PROGRAM MAIN
VAR CONSTANT
	iSoftMajorVersion			: INT	:= 2;
	iSoftMinorVersion			: INT	:= 0;

END_VAR
VAR PERSISTENT
	sMachineCnt					: TprodCounter;
	asStickData					: ARRAY[0..1] OF TStickData;
	asStickDataMMI				: ARRAY[0..1] OF TStickDataMMI;
	sStickDataShared			: TStickDataShared;
	sVacuumSettingsMMI			: TVacuumSettingsMMI;
	TAutoSampling				: TAutoSampling;
	bDisableCleanAfterPearling	: BOOL;
	bDisableVision				: BOOL;
	bSpeedModeSlow				: BOOL;
	iMachineWO					: DINT;
	iMachineSN					: INT;
END_VAR
VAR
	sMMI_SyncVar 				: TMachineData;			(* MMI interface data *)
	sMMI_ManualVar 				: TManualData;			(* MMI interface data for manual mode *)
	sMMI_VisionVar				: TVisionData;			(* Vision interface *)
	sMMI_ConfigFileData			: TConfigFileData;
	(* Blocks definitions *)
	TManager					: Manager;
	TLoaderHandler				: LoaderHdl;
	TTableHandler				: TableHdl;
	TPearlingHandler			: PearlingHdl;
	TSharpenHandler				: SharpenHdl;
	TTurnOverHandler			: TurnOverHdl;
	TBarrelHandler				: BarrelHdl;
	TLift1Handler				: LiftHdl;
	TLift2Handler				: LiftHdl;
	TRejectHandler				: RejectHdl;
	TVisionHandler				: VisionHdl;
	TUtilitiesHandler			: UtilitiesHdl;
	eBarrelCmd					: TModuleCommands;
	eLoaderCmd					: TModuleCommands;
	eTableCmd					: TModuleCommands;
	ePearlingCmd				: TModuleCommands;
	eSharpenCmd					: TModuleCommands;
	eTurnOverCmd				: TModuleCommands;
	eLift1Cmd					: TModuleCommands;
	eLift2Cmd					: TModuleCommands;
	eRejectCmd					: TModuleCommands;
	eVisionCmd					: TModuleCommands;
	eUtilitiesCmd				: TModuleCommands;
	TCheckDoors					: TON;
	sGiversTakers				: TStationGiversTakers;
	bFirstCycle					: BOOL				:= TRUE;
	bJobInProgress				: BOOL;
	bPearlingReady4ChangeTool	: BOOL;
	iStickArea2Use				: INT;
	bTableVacuuumNotOk			: BOOL;
	bPearlingHead1IsUsed		: BOOL;
	bPearlingHead2IsUsed		: BOOL;
	eTableSideForLoader			: TTableSide;
	sRunData					: TRunData;
	bTableAspiration13On		: BOOL;
	bTableAspiration24On		: BOOL;
	bLoaderBrushAspirationOn	: BOOL;
	bBrushAspirationOn			: BOOL;
	bSharpenAspirationOn		: BOOL;
	bStopRequest				: BOOL;
	bPauseRequest				: BOOL;
	bLayeringWithTwoParts		: BOOL;
	bNewPlateLift1				: BOOL;
	bNewPlateLift2				: BOOL;
	bNewPlateReject				: BOOL;
	bLoaderVacuumInUse			: BOOL;
	bManInterlockPearling		: BOOL;
	bManInterlockLoader			: BOOL;
	bManInterlockLoaderLift		: BOOL;
	bManInterlockTable			: BOOL;
	bManInterlockTurnOver		: BOOL;
	TJobElapsed					: TIME;
	aiTablePearlsVacuumFlow		: ARRAY[0..1] OF INT;
END_VAR
VAR // added by the converter: edge detectors and wires of the graphical bodies
    _w1, _w3 : TStickData;
    _w2, _w4 : TStickDataMMI;
    _w5 : TStickDataMMIShared;
    _w6 : TVacuumSettingsMMI;
    _w7 : TprodCounter;
    _w8, _w9, _w11, _w12 : INT;
    _w10, _w13, _w14, _w15 : BOOL;
END_VAR

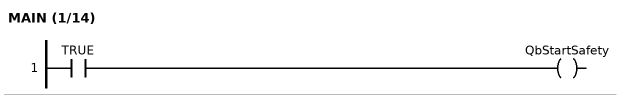
// NETWORK 1
QbStartSafety := TRUE;

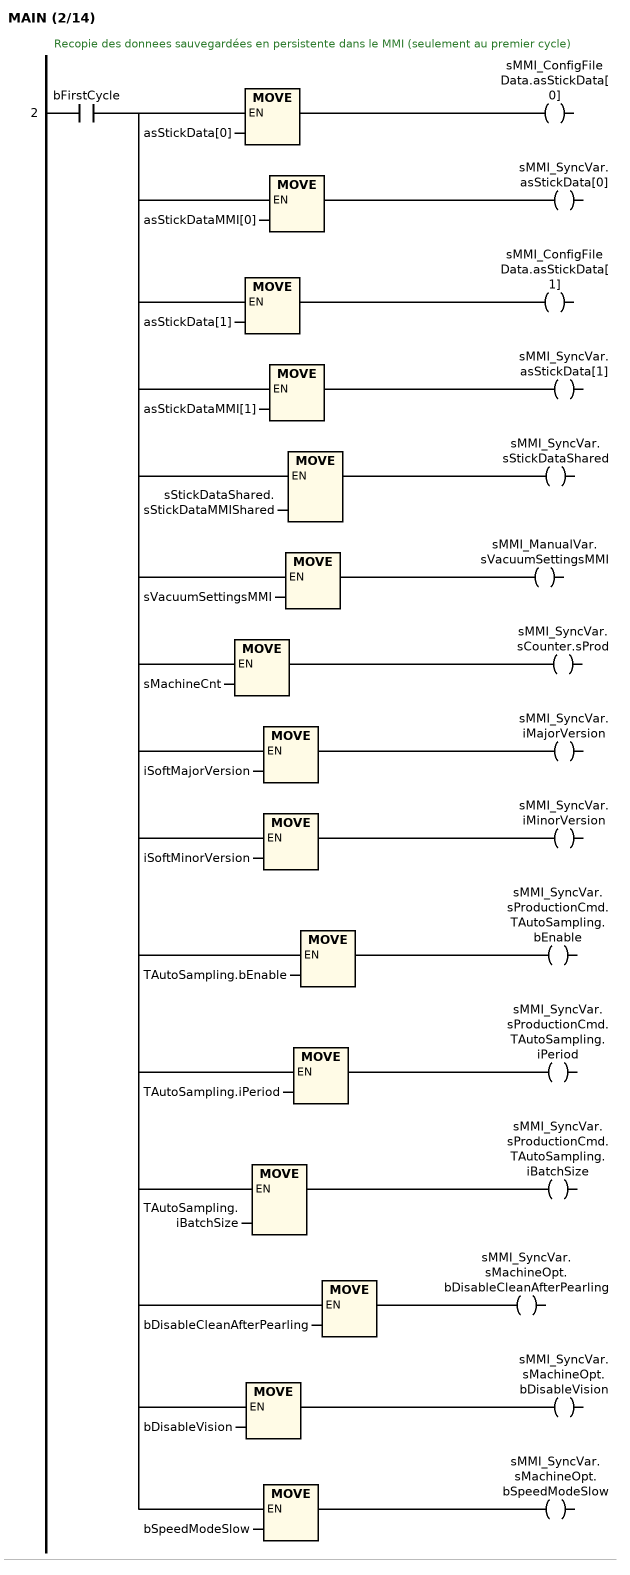
// NETWORK 2
// Recopie des donnees sauvegardées en persistente dans le MMI (seulement au premier cycle)
IF bFirstCycle THEN _w1 := asStickData[0]; END_IF
sMMI_ConfigFileData.asStickData[0] := _w1;
IF bFirstCycle THEN _w2 := asStickDataMMI[0]; END_IF
sMMI_SyncVar.asStickData[0] := _w2;
IF bFirstCycle THEN _w3 := asStickData[1]; END_IF
sMMI_ConfigFileData.asStickData[1] := _w3;
IF bFirstCycle THEN _w4 := asStickDataMMI[1]; END_IF
sMMI_SyncVar.asStickData[1] := _w4;
IF bFirstCycle THEN _w5 := sStickDataShared.sStickDataMMIShared; END_IF
sMMI_SyncVar.sStickDataShared := _w5;
IF bFirstCycle THEN _w6 := sVacuumSettingsMMI; END_IF
sMMI_ManualVar.sVacuumSettingsMMI := _w6;
IF bFirstCycle THEN _w7 := sMachineCnt; END_IF
sMMI_SyncVar.sCounter.sProd := _w7;
IF bFirstCycle THEN _w8 := iSoftMajorVersion; END_IF
sMMI_SyncVar.iMajorVersion := _w8;
IF bFirstCycle THEN _w9 := iSoftMinorVersion; END_IF
sMMI_SyncVar.iMinorVersion := _w9;
IF bFirstCycle THEN _w10 := TAutoSampling.bEnable; END_IF
sMMI_SyncVar.sProductionCmd.TAutoSampling.bEnable := _w10;
IF bFirstCycle THEN _w11 := TAutoSampling.iPeriod; END_IF
sMMI_SyncVar.sProductionCmd.TAutoSampling.iPeriod := _w11;
IF bFirstCycle THEN _w12 := TAutoSampling.iBatchSize; END_IF
sMMI_SyncVar.sProductionCmd.TAutoSampling.iBatchSize := _w12;
IF bFirstCycle THEN _w13 := bDisableCleanAfterPearling; END_IF
sMMI_SyncVar.sMachineOpt.bDisableCleanAfterPearling := _w13;
IF bFirstCycle THEN _w14 := bDisableVision; END_IF
sMMI_SyncVar.sMachineOpt.bDisableVision := _w14;
IF bFirstCycle THEN _w15 := bSpeedModeSlow; END_IF
sMMI_SyncVar.sMachineOpt.bSpeedModeSlow := _w15;

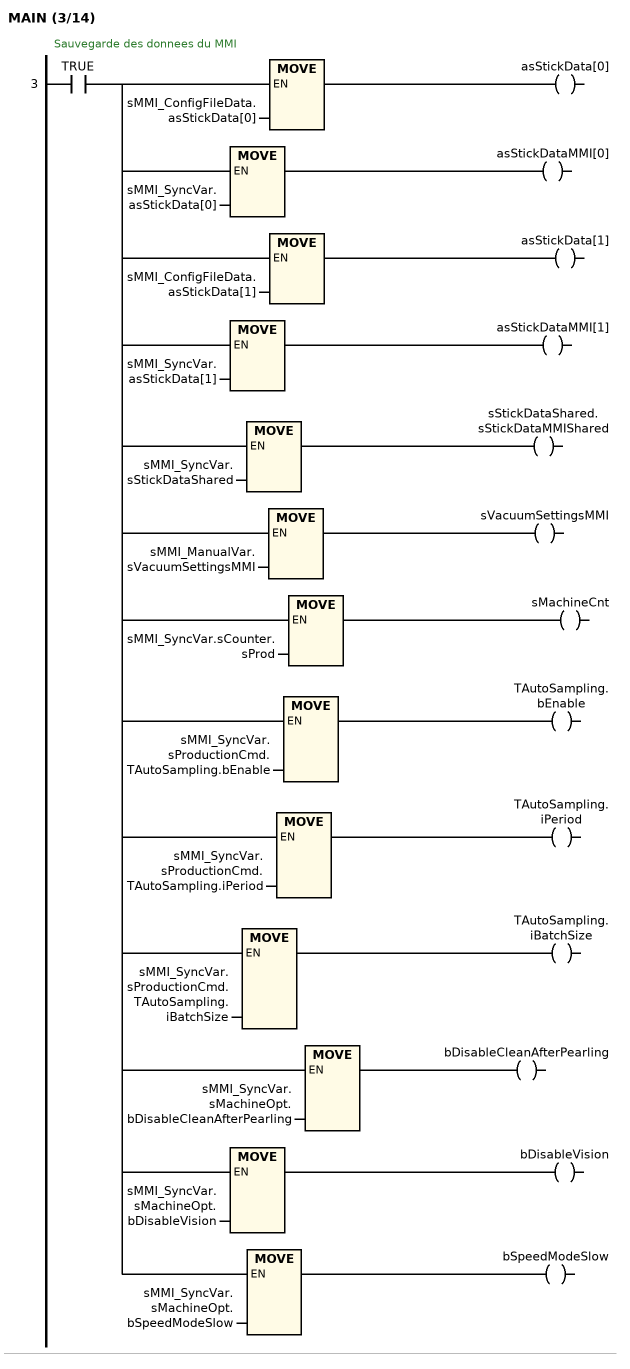
// NETWORK 3
// Sauvegarde des donnees du MMI
asStickData[0] := sMMI_ConfigFileData.asStickData[0];
asStickDataMMI[0] := sMMI_SyncVar.asStickData[0];
asStickData[1] := sMMI_ConfigFileData.asStickData[1];
asStickDataMMI[1] := sMMI_SyncVar.asStickData[1];
sStickDataShared.sStickDataMMIShared := sMMI_SyncVar.sStickDataShared;
sVacuumSettingsMMI := sMMI_ManualVar.sVacuumSettingsMMI;
sMachineCnt := sMMI_SyncVar.sCounter.sProd;
TAutoSampling.bEnable := sMMI_SyncVar.sProductionCmd.TAutoSampling.bEnable;
TAutoSampling.iPeriod := sMMI_SyncVar.sProductionCmd.TAutoSampling.iPeriod;
TAutoSampling.iBatchSize := sMMI_SyncVar.sProductionCmd.TAutoSampling.iBatchSize;
bDisableCleanAfterPearling := sMMI_SyncVar.sMachineOpt.bDisableCleanAfterPearling;
bDisableVision := sMMI_SyncVar.sMachineOpt.bDisableVision;
bSpeedModeSlow := sMMI_SyncVar.sMachineOpt.bSpeedModeSlow;

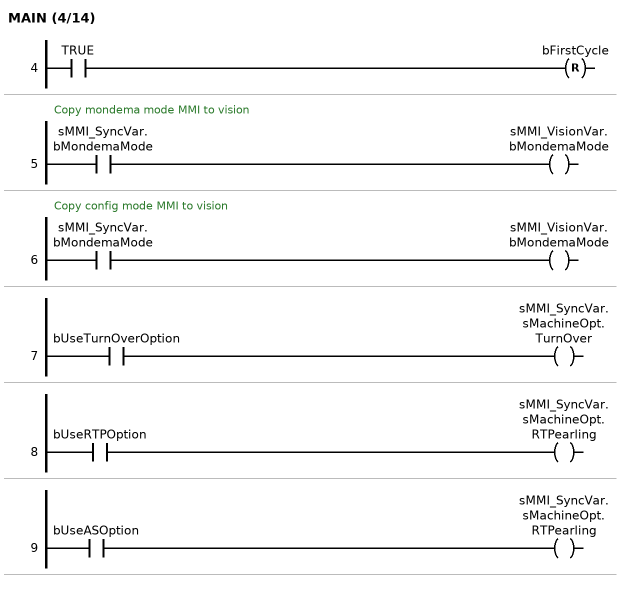
// NETWORK 4
bFirstCycle R= TRUE;

// NETWORK 5
// Copy mondema mode MMI to vision
sMMI_VisionVar.bMondemaMode := sMMI_SyncVar.bMondemaMode;

// NETWORK 6
// Copy config mode MMI to vision
sMMI_VisionVar.bMondemaMode := sMMI_SyncVar.bMondemaMode;

// NETWORK 7
sMMI_SyncVar.sMachineOpt.TurnOver := bUseTurnOverOption;

// NETWORK 8
sMMI_SyncVar.sMachineOpt.RTPearling := bUseRTPOption;

// NETWORK 9
sMMI_SyncVar.sMachineOpt.RTPearling := bUseASOption;

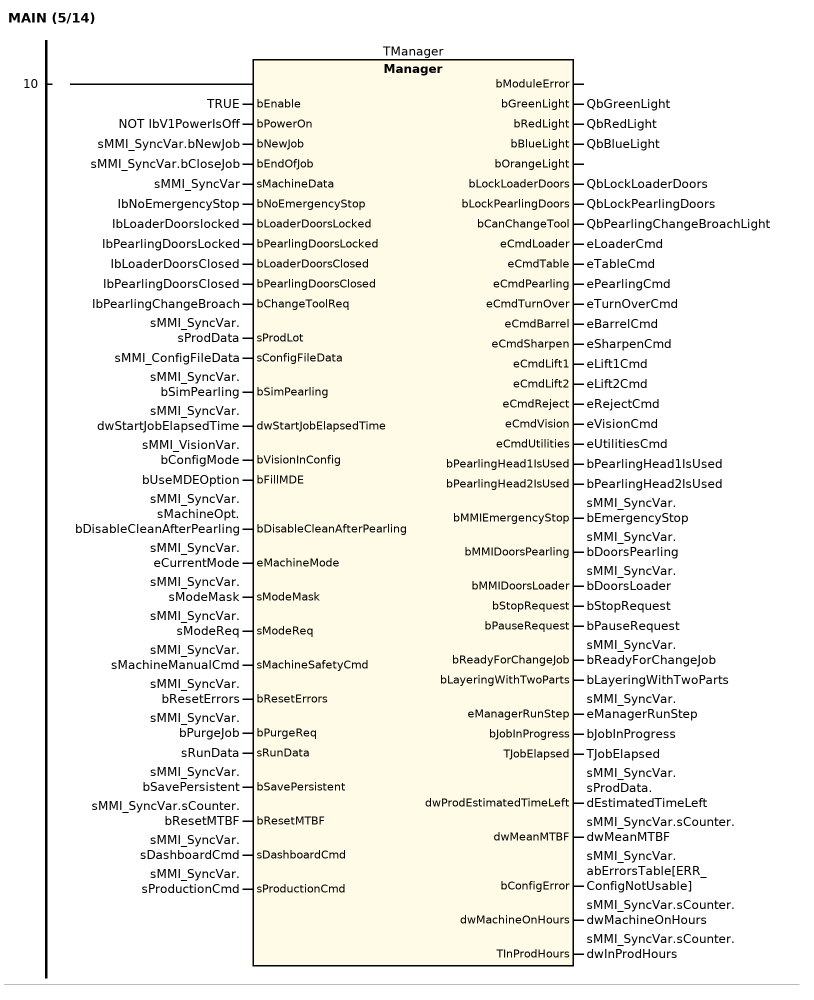
// NETWORK 10
TManager(
    bEnable := TRUE,
    bPowerOn := NOT IbV1PowerIsOff,
    bNewJob := sMMI_SyncVar.bNewJob,
    bEndOfJob := sMMI_SyncVar.bCloseJob,
    sMachineData := sMMI_SyncVar,
    bNoEmergencyStop := IbNoEmergencyStop,
    bLoaderDoorsLocked := IbLoaderDoorslocked,
    bPearlingDoorsLocked := IbPearlingDoorsLocked,
    bLoaderDoorsClosed := IbLoaderDoorsClosed,
    bPearlingDoorsClosed := IbPearlingDoorsClosed,
    bChangeToolReq := IbPearlingChangeBroach,
    sProdLot := sMMI_SyncVar.sProdData,
    sConfigFileData := sMMI_ConfigFileData,
    bSimPearling := sMMI_SyncVar.bSimPearling,
    dwStartJobElapsedTime := sMMI_SyncVar.dwStartJobElapsedTime,
    bVisionInConfig := sMMI_VisionVar.bConfigMode,
    bFillMDE := bUseMDEOption,
    bDisableCleanAfterPearling := sMMI_SyncVar.sMachineOpt.bDisableCleanAfterPearling,
    eMachineMode := sMMI_SyncVar.eCurrentMode,
    sModeMask := sMMI_SyncVar.sModeMask,
    sModeReq := sMMI_SyncVar.sModeReq,
    sMachineSafetyCmd := sMMI_SyncVar.sMachineManualCmd,
    bResetErrors := sMMI_SyncVar.bResetErrors,
    bPurgeReq := sMMI_SyncVar.bPurgeJob,
    sRunData := sRunData,
    bSavePersistent := sMMI_SyncVar.bSavePersistent,
    bResetMTBF := sMMI_SyncVar.sCounter.bResetMTBF,
    sDashboardCmd := sMMI_SyncVar.sDashboardCmd,
    sProductionCmd := sMMI_SyncVar.sProductionCmd,
    bGreenLight => QbGreenLight,
    bRedLight => QbRedLight,
    bBlueLight => QbBlueLight,
    bLockLoaderDoors => QbLockLoaderDoors,
    bLockPearlingDoors => QbLockPearlingDoors,
    bCanChangeTool => QbPearlingChangeBroachLight,
    eCmdLoader => eLoaderCmd,
    eCmdTable => eTableCmd,
    eCmdPearling => ePearlingCmd,
    eCmdTurnOver => eTurnOverCmd,
    eCmdBarrel => eBarrelCmd,
    eCmdSharpen => eSharpenCmd,
    eCmdLift1 => eLift1Cmd,
    eCmdLift2 => eLift2Cmd,
    eCmdReject => eRejectCmd,
    eCmdVision => eVisionCmd,
    eCmdUtilities => eUtilitiesCmd,
    bPearlingHead1IsUsed => bPearlingHead1IsUsed,
    bPearlingHead2IsUsed => bPearlingHead2IsUsed,
    bMMIEmergencyStop => sMMI_SyncVar.bEmergencyStop,
    bMMIDoorsPearling => sMMI_SyncVar.bDoorsPearling,
    bMMIDoorsLoader => sMMI_SyncVar.bDoorsLoader,
    bStopRequest => bStopRequest,
    bPauseRequest => bPauseRequest,
    bReadyForChangeJob => sMMI_SyncVar.bReadyForChangeJob,
    bLayeringWithTwoParts => bLayeringWithTwoParts,
    eManagerRunStep => sMMI_SyncVar.eManagerRunStep,
    bJobInProgress => bJobInProgress,
    TJobElapsed => TJobElapsed,
    dwProdEstimatedTimeLeft => sMMI_SyncVar.sProdData.dEstimatedTimeLeft,
    dwMeanMTBF => sMMI_SyncVar.sCounter.dwMeanMTBF,
    bConfigError => sMMI_SyncVar.abErrorsTable[ERR_ConfigNotUsable],
    dwMachineOnHours => sMMI_SyncVar.sCounter.dwMachineOnHours,
    TInProdHours => sMMI_SyncVar.sCounter.dwInProdHours); // Manager

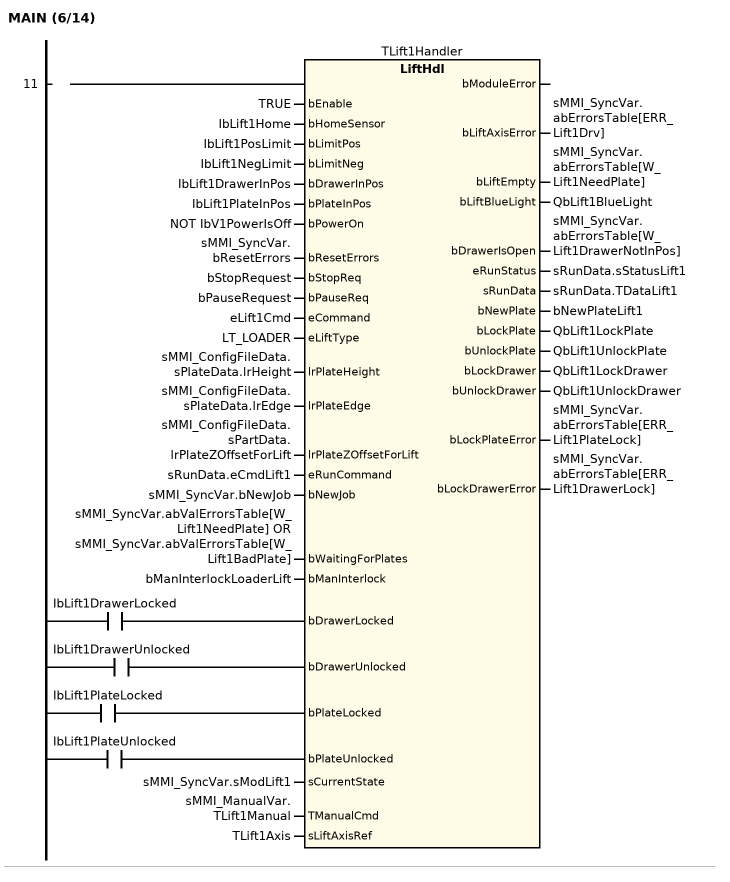
// NETWORK 11
TLift1Handler(
    bEnable := TRUE,
    bHomeSensor := IbLift1Home,
    bLimitPos := IbLift1PosLimit,
    bLimitNeg := IbLift1NegLimit,
    bDrawerInPos := IbLift1DrawerInPos,
    bPlateInPos := IbLift1PlateInPos,
    bPowerOn := NOT IbV1PowerIsOff,
    bResetErrors := sMMI_SyncVar.bResetErrors,
    bStopReq := bStopRequest,
    bPauseReq := bPauseRequest,
    eCommand := eLift1Cmd,
    eLiftType := LT_LOADER,
    lrPlateHeight := sMMI_ConfigFileData.sPlateData.lrHeight,
    lrPlateEdge := sMMI_ConfigFileData.sPlateData.lrEdge,
    lrPlateZOffsetForLift := sMMI_ConfigFileData.sPartData.lrPlateZOffsetForLift,
    eRunCommand := sRunData.eCmdLift1,
    bNewJob := sMMI_SyncVar.bNewJob,
    bWaitingForPlates := sMMI_SyncVar.abValErrorsTable[W_Lift1NeedPlate] OR sMMI_SyncVar.abValErrorsTable[W_Lift1BadPlate],
    bManInterlock := bManInterlockLoaderLift,
    bDrawerLocked := IbLift1DrawerLocked,
    bDrawerUnlocked := IbLift1DrawerUnlocked,
    bPlateLocked := IbLift1PlateLocked,
    bPlateUnlocked := IbLift1PlateUnlocked,
    sCurrentState := sMMI_SyncVar.sModLift1,
    TManualCmd := sMMI_ManualVar.TLift1Manual,
    sLiftAxisRef := TLift1Axis,
    bLiftAxisError => sMMI_SyncVar.abErrorsTable[ERR_Lift1Drv],
    bLiftEmpty => sMMI_SyncVar.abErrorsTable[W_Lift1NeedPlate],
    bLiftBlueLight => QbLift1BlueLight,
    bDrawerIsOpen => sMMI_SyncVar.abErrorsTable[W_Lift1DrawerNotInPos],
    eRunStatus => sRunData.sStatusLift1,
    sRunData => sRunData.TDataLift1,
    bNewPlate => bNewPlateLift1,
    bLockPlate => QbLift1LockPlate,
    bUnlockPlate => QbLift1UnlockPlate,
    bLockDrawer => QbLift1LockDrawer,
    bUnlockDrawer => QbLift1UnlockDrawer,
    bLockPlateError => sMMI_SyncVar.abErrorsTable[ERR_Lift1PlateLock],
    bLockDrawerError => sMMI_SyncVar.abErrorsTable[ERR_Lift1DrawerLock]); // LiftHdl

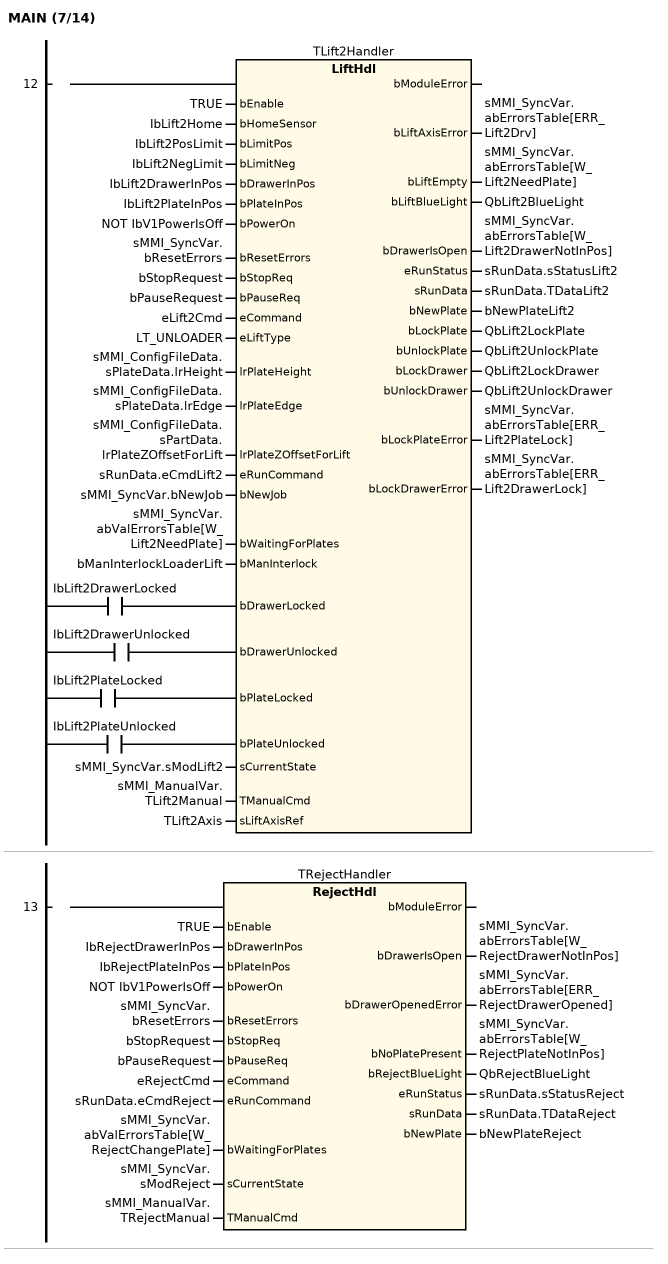
// NETWORK 12
TLift2Handler(
    bEnable := TRUE,
    bHomeSensor := IbLift2Home,
    bLimitPos := IbLift2PosLimit,
    bLimitNeg := IbLift2NegLimit,
    bDrawerInPos := IbLift2DrawerInPos,
    bPlateInPos := IbLift2PlateInPos,
    bPowerOn := NOT IbV1PowerIsOff,
    bResetErrors := sMMI_SyncVar.bResetErrors,
    bStopReq := bStopRequest,
    bPauseReq := bPauseRequest,
    eCommand := eLift2Cmd,
    eLiftType := LT_UNLOADER,
    lrPlateHeight := sMMI_ConfigFileData.sPlateData.lrHeight,
    lrPlateEdge := sMMI_ConfigFileData.sPlateData.lrEdge,
    lrPlateZOffsetForLift := sMMI_ConfigFileData.sPartData.lrPlateZOffsetForLift,
    eRunCommand := sRunData.eCmdLift2,
    bNewJob := sMMI_SyncVar.bNewJob,
    bWaitingForPlates := sMMI_SyncVar.abValErrorsTable[W_Lift2NeedPlate],
    bManInterlock := bManInterlockLoaderLift,
    bDrawerLocked := IbLift2DrawerLocked,
    bDrawerUnlocked := IbLift2DrawerUnlocked,
    bPlateLocked := IbLift2PlateLocked,
    bPlateUnlocked := IbLift2PlateUnlocked,
    sCurrentState := sMMI_SyncVar.sModLift2,
    TManualCmd := sMMI_ManualVar.TLift2Manual,
    sLiftAxisRef := TLift2Axis,
    bLiftAxisError => sMMI_SyncVar.abErrorsTable[ERR_Lift2Drv],
    bLiftEmpty => sMMI_SyncVar.abErrorsTable[W_Lift2NeedPlate],
    bLiftBlueLight => QbLift2BlueLight,
    bDrawerIsOpen => sMMI_SyncVar.abErrorsTable[W_Lift2DrawerNotInPos],
    eRunStatus => sRunData.sStatusLift2,
    sRunData => sRunData.TDataLift2,
    bNewPlate => bNewPlateLift2,
    bLockPlate => QbLift2LockPlate,
    bUnlockPlate => QbLift2UnlockPlate,
    bLockDrawer => QbLift2LockDrawer,
    bUnlockDrawer => QbLift2UnlockDrawer,
    bLockPlateError => sMMI_SyncVar.abErrorsTable[ERR_Lift2PlateLock],
    bLockDrawerError => sMMI_SyncVar.abErrorsTable[ERR_Lift2DrawerLock]); // LiftHdl

// NETWORK 13
TRejectHandler(
    bEnable := TRUE,
    bDrawerInPos := IbRejectDrawerInPos,
    bPlateInPos := IbRejectPlateInPos,
    bPowerOn := NOT IbV1PowerIsOff,
    bResetErrors := sMMI_SyncVar.bResetErrors,
    bStopReq := bStopRequest,
    bPauseReq := bPauseRequest,
    eCommand := eRejectCmd,
    eRunCommand := sRunData.eCmdReject,
    bWaitingForPlates := sMMI_SyncVar.abValErrorsTable[W_RejectChangePlate],
    sCurrentState := sMMI_SyncVar.sModReject,
    TManualCmd := sMMI_ManualVar.TRejectManual,
    bDrawerIsOpen => sMMI_SyncVar.abErrorsTable[W_RejectDrawerNotInPos],
    bDrawerOpenedError => sMMI_SyncVar.abErrorsTable[ERR_RejectDrawerOpened],
    bNoPlatePresent => sMMI_SyncVar.abErrorsTable[W_RejectPlateNotInPos],
    bRejectBlueLight => QbRejectBlueLight,
    eRunStatus => sRunData.sStatusReject,
    sRunData => sRunData.TDataReject,
    bNewPlate => bNewPlateReject); // RejectHdl

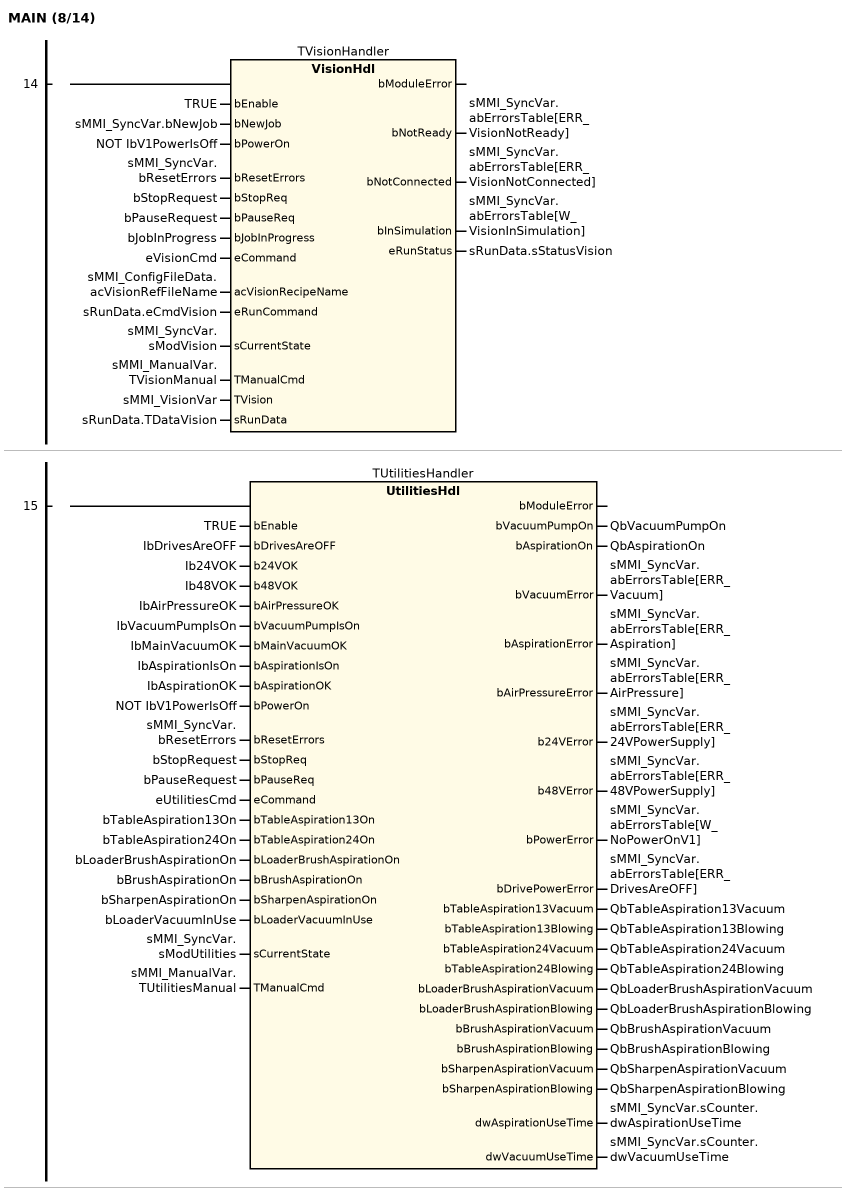
// NETWORK 14
TVisionHandler(
    bEnable := TRUE,
    bNewJob := sMMI_SyncVar.bNewJob,
    bPowerOn := NOT IbV1PowerIsOff,
    bResetErrors := sMMI_SyncVar.bResetErrors,
    bStopReq := bStopRequest,
    bPauseReq := bPauseRequest,
    bJobInProgress := bJobInProgress,
    eCommand := eVisionCmd,
    acVisionRecipeName := sMMI_ConfigFileData.acVisionRefFileName,
    eRunCommand := sRunData.eCmdVision,
    sCurrentState := sMMI_SyncVar.sModVision,
    TManualCmd := sMMI_ManualVar.TVisionManual,
    TVision := sMMI_VisionVar,
    sRunData := sRunData.TDataVision,
    bNotReady => sMMI_SyncVar.abErrorsTable[ERR_VisionNotReady],
    bNotConnected => sMMI_SyncVar.abErrorsTable[ERR_VisionNotConnected],
    bInSimulation => sMMI_SyncVar.abErrorsTable[W_VisionInSimulation],
    eRunStatus => sRunData.sStatusVision); // VisionHdl

// NETWORK 15
TUtilitiesHandler(
    bEnable := TRUE,
    bDrivesAreOFF := IbDrivesAreOFF,
    b24VOK := Ib24VOK,
    b48VOK := Ib48VOK,
    bAirPressureOK := IbAirPressureOK,
    bVacuumPumpIsOn := IbVacuumPumpIsOn,
    bMainVacuumOK := IbMainVacuumOK,
    bAspirationIsOn := IbAspirationIsOn,
    bAspirationOK := IbAspirationOK,
    bPowerOn := NOT IbV1PowerIsOff,
    bResetErrors := sMMI_SyncVar.bResetErrors,
    bStopReq := bStopRequest,
    bPauseReq := bPauseRequest,
    eCommand := eUtilitiesCmd,
    bTableAspiration13On := bTableAspiration13On,
    bTableAspiration24On := bTableAspiration24On,
    bLoaderBrushAspirationOn := bLoaderBrushAspirationOn,
    bBrushAspirationOn := bBrushAspirationOn,
    bSharpenAspirationOn := bSharpenAspirationOn,
    bLoaderVacuumInUse := bLoaderVacuumInUse,
    sCurrentState := sMMI_SyncVar.sModUtilities,
    TManualCmd := sMMI_ManualVar.TUtilitiesManual,
    bVacuumPumpOn => QbVacuumPumpOn,
    bAspirationOn => QbAspirationOn,
    bVacuumError => sMMI_SyncVar.abErrorsTable[ERR_Vacuum],
    bAspirationError => sMMI_SyncVar.abErrorsTable[ERR_Aspiration],
    bAirPressureError => sMMI_SyncVar.abErrorsTable[ERR_AirPressure],
    b24VError => sMMI_SyncVar.abErrorsTable[ERR_24VPowerSupply],
    b48VError => sMMI_SyncVar.abErrorsTable[ERR_48VPowerSupply],
    bPowerError => sMMI_SyncVar.abErrorsTable[W_NoPowerOnV1],
    bDrivePowerError => sMMI_SyncVar.abErrorsTable[ERR_DrivesAreOFF],
    bTableAspiration13Vacuum => QbTableAspiration13Vacuum,
    bTableAspiration13Blowing => QbTableAspiration13Blowing,
    bTableAspiration24Vacuum => QbTableAspiration24Vacuum,
    bTableAspiration24Blowing => QbTableAspiration24Blowing,
    bLoaderBrushAspirationVacuum => QbLoaderBrushAspirationVacuum,
    bLoaderBrushAspirationBlowing => QbLoaderBrushAspirationBlowing,
    bBrushAspirationVacuum => QbBrushAspirationVacuum,
    bBrushAspirationBlowing => QbBrushAspirationBlowing,
    bSharpenAspirationVacuum => QbSharpenAspirationVacuum,
    bSharpenAspirationBlowing => QbSharpenAspirationBlowing,
    dwAspirationUseTime => sMMI_SyncVar.sCounter.dwAspirationUseTime,
    dwVacuumUseTime => sMMI_SyncVar.sCounter.dwVacuumUseTime); // UtilitiesHdl

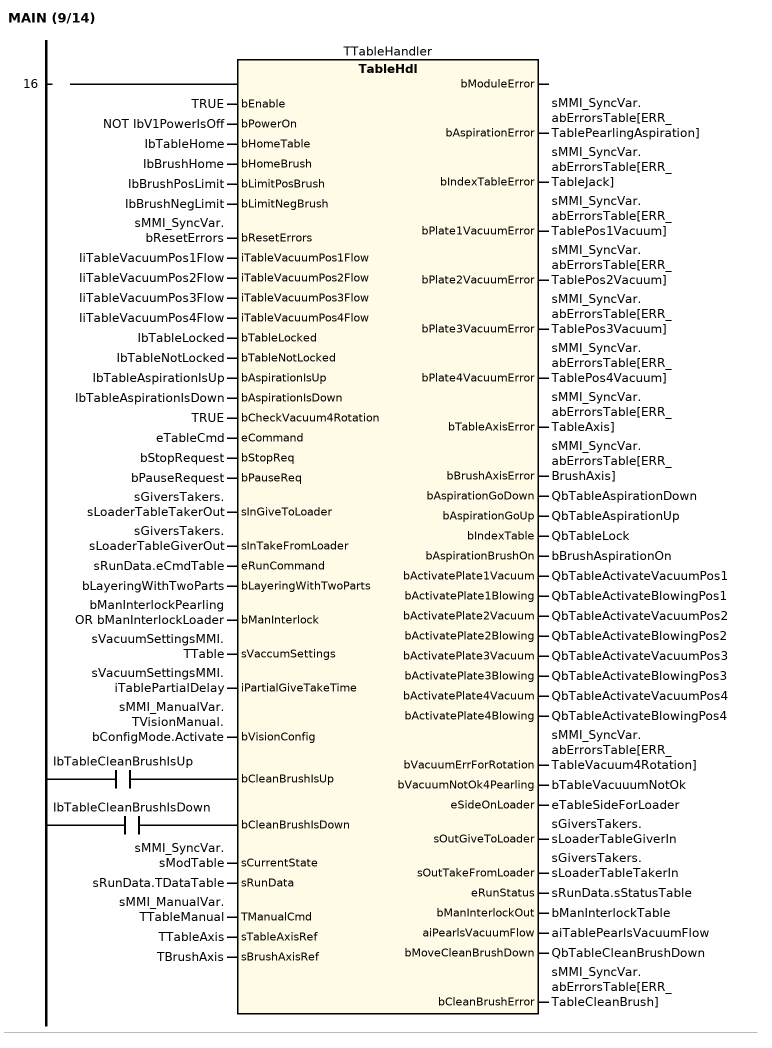
// NETWORK 16
TTableHandler(
    bEnable := TRUE,
    bPowerOn := NOT IbV1PowerIsOff,
    bHomeTable := IbTableHome,
    bHomeBrush := IbBrushHome,
    bLimitPosBrush := IbBrushPosLimit,
    bLimitNegBrush := IbBrushNegLimit,
    bResetErrors := sMMI_SyncVar.bResetErrors,
    iTableVacuumPos1Flow := IiTableVacuumPos1Flow,
    iTableVacuumPos2Flow := IiTableVacuumPos2Flow,
    iTableVacuumPos3Flow := IiTableVacuumPos3Flow,
    iTableVacuumPos4Flow := IiTableVacuumPos4Flow,
    bTableLocked := IbTableLocked,
    bTableNotLocked := IbTableNotLocked,
    bAspirationIsUp := IbTableAspirationIsUp,
    bAspirationIsDown := IbTableAspirationIsDown,
    bCheckVacuum4Rotation := TRUE,
    eCommand := eTableCmd,
    bStopReq := bStopRequest,
    bPauseReq := bPauseRequest,
    sInGiveToLoader := sGiversTakers.sLoaderTableTakerOut,
    sInTakeFromLoader := sGiversTakers.sLoaderTableGiverOut,
    eRunCommand := sRunData.eCmdTable,
    bLayeringWithTwoParts := bLayeringWithTwoParts,
    bManInterlock := bManInterlockPearling OR bManInterlockLoader,
    sVaccumSettings := sVacuumSettingsMMI.TTable,
    iPartialGiveTakeTime := sVacuumSettingsMMI.iTablePartialDelay,
    bVisionConfig := sMMI_ManualVar.TVisionManual.bConfigMode.Activate,
    bCleanBrushIsUp := IbTableCleanBrushIsUp,
    bCleanBrushIsDown := IbTableCleanBrushIsDown,
    sCurrentState := sMMI_SyncVar.sModTable,
    sRunData := sRunData.TDataTable,
    TManualCmd := sMMI_ManualVar.TTableManual,
    sTableAxisRef := TTableAxis,
    sBrushAxisRef := TBrushAxis,
    bAspirationError => sMMI_SyncVar.abErrorsTable[ERR_TablePearlingAspiration],
    bIndexTableError => sMMI_SyncVar.abErrorsTable[ERR_TableJack],
    bPlate1VacuumError => sMMI_SyncVar.abErrorsTable[ERR_TablePos1Vacuum],
    bPlate2VacuumError => sMMI_SyncVar.abErrorsTable[ERR_TablePos2Vacuum],
    bPlate3VacuumError => sMMI_SyncVar.abErrorsTable[ERR_TablePos3Vacuum],
    bPlate4VacuumError => sMMI_SyncVar.abErrorsTable[ERR_TablePos4Vacuum],
    bTableAxisError => sMMI_SyncVar.abErrorsTable[ERR_TableAxis],
    bBrushAxisError => sMMI_SyncVar.abErrorsTable[ERR_BrushAxis],
    bAspirationGoDown => QbTableAspirationDown,
    bAspirationGoUp => QbTableAspirationUp,
    bIndexTable => QbTableLock,
    bAspirationBrushOn => bBrushAspirationOn,
    bActivatePlate1Vacuum => QbTableActivateVacuumPos1,
    bActivatePlate1Blowing => QbTableActivateBlowingPos1,
    bActivatePlate2Vacuum => QbTableActivateVacuumPos2,
    bActivatePlate2Blowing => QbTableActivateBlowingPos2,
    bActivatePlate3Vacuum => QbTableActivateVacuumPos3,
    bActivatePlate3Blowing => QbTableActivateBlowingPos3,
    bActivatePlate4Vacuum => QbTableActivateVacuumPos4,
    bActivatePlate4Blowing => QbTableActivateBlowingPos4,
    bVacuumErrForRotation => sMMI_SyncVar.abErrorsTable[ERR_TableVacuum4Rotation],
    bVacuumNotOk4Pearling => bTableVacuuumNotOk,
    eSideOnLoader => eTableSideForLoader,
    sOutGiveToLoader => sGiversTakers.sLoaderTableGiverIn,
    sOutTakeFromLoader => sGiversTakers.sLoaderTableTakerIn,
    eRunStatus => sRunData.sStatusTable,
    bManInterlockOut => bManInterlockTable,
    aiPearlsVacuumFlow => aiTablePearlsVacuumFlow,
    bMoveCleanBrushDown => QbTableCleanBrushDown,
    bCleanBrushError => sMMI_SyncVar.abErrorsTable[ERR_TableCleanBrush]); // TableHdl

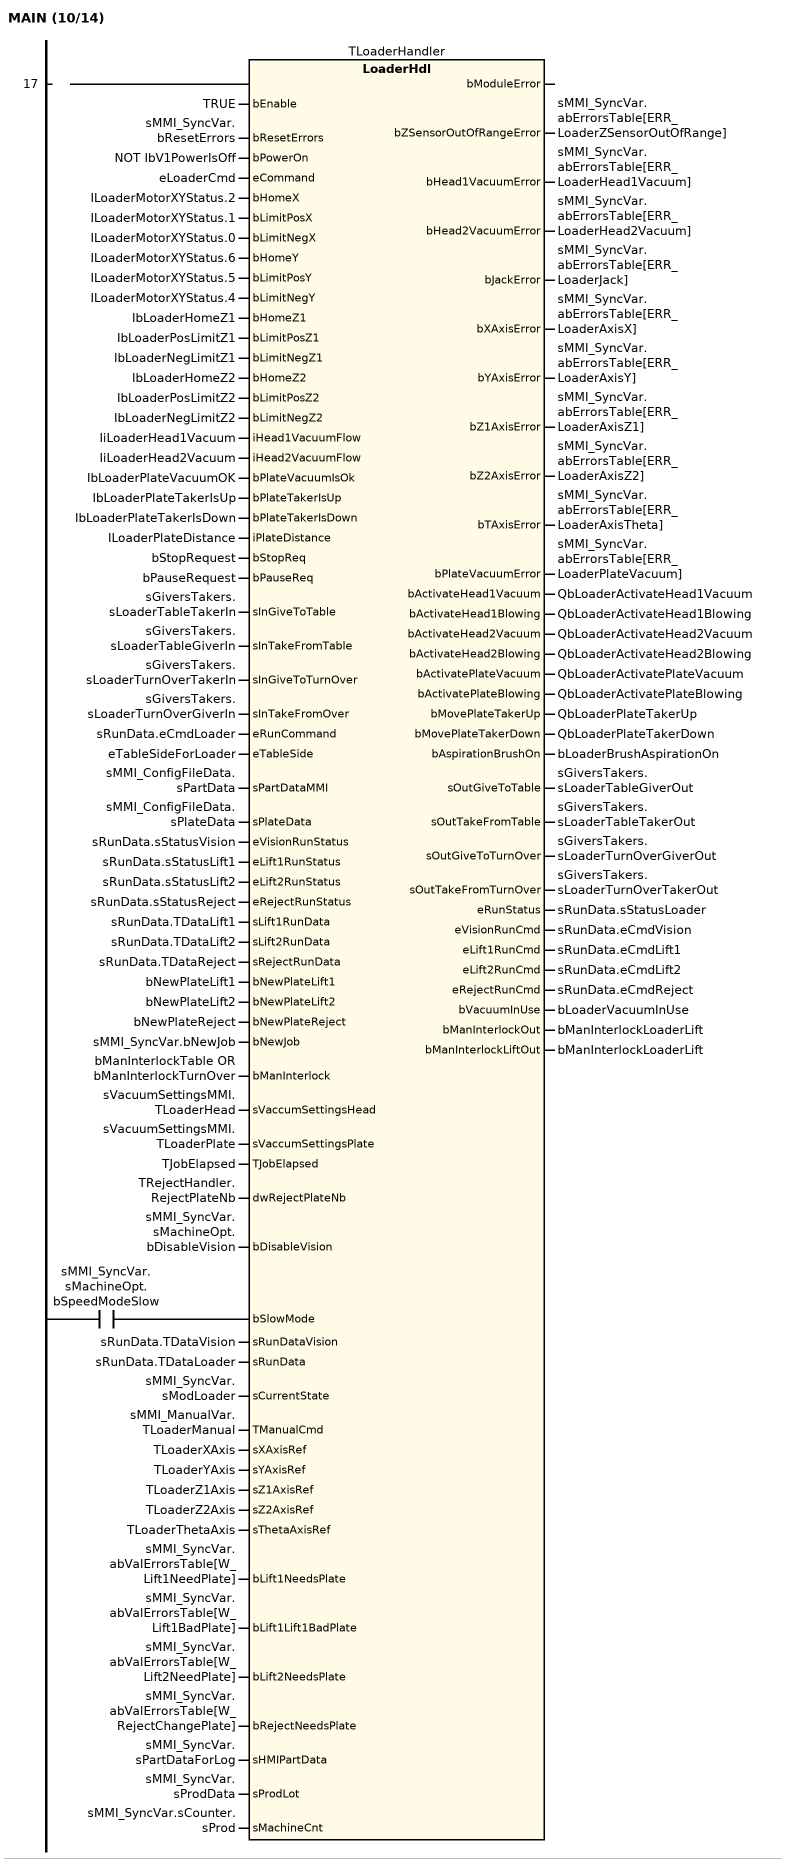
// NETWORK 17
TLoaderHandler(
    bEnable := TRUE,
    bResetErrors := sMMI_SyncVar.bResetErrors,
    bPowerOn := NOT IbV1PowerIsOff,
    eCommand := eLoaderCmd,
    bHomeX := ILoaderMotorXYStatus.2,
    bLimitPosX := ILoaderMotorXYStatus.1,
    bLimitNegX := ILoaderMotorXYStatus.0,
    bHomeY := ILoaderMotorXYStatus.6,
    bLimitPosY := ILoaderMotorXYStatus.5,
    bLimitNegY := ILoaderMotorXYStatus.4,
    bHomeZ1 := IbLoaderHomeZ1,
    bLimitPosZ1 := IbLoaderPosLimitZ1,
    bLimitNegZ1 := IbLoaderNegLimitZ1,
    bHomeZ2 := IbLoaderHomeZ2,
    bLimitPosZ2 := IbLoaderPosLimitZ2,
    bLimitNegZ2 := IbLoaderNegLimitZ2,
    iHead1VacuumFlow := IiLoaderHead1Vacuum,
    iHead2VacuumFlow := IiLoaderHead2Vacuum,
    bPlateVacuumIsOk := IbLoaderPlateVacuumOK,
    bPlateTakerIsUp := IbLoaderPlateTakerIsUp,
    bPlateTakerIsDown := IbLoaderPlateTakerIsDown,
    iPlateDistance := ILoaderPlateDistance,
    bStopReq := bStopRequest,
    bPauseReq := bPauseRequest,
    sInGiveToTable := sGiversTakers.sLoaderTableTakerIn,
    sInTakeFromTable := sGiversTakers.sLoaderTableGiverIn,
    sInGiveToTurnOver := sGiversTakers.sLoaderTurnOverTakerIn,
    sInTakeFromOver := sGiversTakers.sLoaderTurnOverGiverIn,
    eRunCommand := sRunData.eCmdLoader,
    eTableSide := eTableSideForLoader,
    sPartDataMMI := sMMI_ConfigFileData.sPartData,
    sPlateData := sMMI_ConfigFileData.sPlateData,
    eVisionRunStatus := sRunData.sStatusVision,
    eLift1RunStatus := sRunData.sStatusLift1,
    eLift2RunStatus := sRunData.sStatusLift2,
    eRejectRunStatus := sRunData.sStatusReject,
    sLift1RunData := sRunData.TDataLift1,
    sLift2RunData := sRunData.TDataLift2,
    sRejectRunData := sRunData.TDataReject,
    bNewPlateLift1 := bNewPlateLift1,
    bNewPlateLift2 := bNewPlateLift2,
    bNewPlateReject := bNewPlateReject,
    bNewJob := sMMI_SyncVar.bNewJob,
    bManInterlock := bManInterlockTable OR bManInterlockTurnOver,
    sVaccumSettingsHead := sVacuumSettingsMMI.TLoaderHead,
    sVaccumSettingsPlate := sVacuumSettingsMMI.TLoaderPlate,
    TJobElapsed := TJobElapsed,
    dwRejectPlateNb := TRejectHandler.RejectPlateNb,
    bDisableVision := sMMI_SyncVar.sMachineOpt.bDisableVision,
    bSlowMode := sMMI_SyncVar.sMachineOpt.bSpeedModeSlow,
    sRunDataVision := sRunData.TDataVision,
    sRunData := sRunData.TDataLoader,
    sCurrentState := sMMI_SyncVar.sModLoader,
    TManualCmd := sMMI_ManualVar.TLoaderManual,
    sXAxisRef := TLoaderXAxis,
    sYAxisRef := TLoaderYAxis,
    sZ1AxisRef := TLoaderZ1Axis,
    sZ2AxisRef := TLoaderZ2Axis,
    sThetaAxisRef := TLoaderThetaAxis,
    bLift1NeedsPlate := sMMI_SyncVar.abValErrorsTable[W_Lift1NeedPlate],
    bLift1Lift1BadPlate := sMMI_SyncVar.abValErrorsTable[W_Lift1BadPlate],
    bLift2NeedsPlate := sMMI_SyncVar.abValErrorsTable[W_Lift2NeedPlate],
    bRejectNeedsPlate := sMMI_SyncVar.abValErrorsTable[W_RejectChangePlate],
    sHMIPartData := sMMI_SyncVar.sPartDataForLog,
    sProdLot := sMMI_SyncVar.sProdData,
    sMachineCnt := sMMI_SyncVar.sCounter.sProd,
    bZSensorOutOfRangeError => sMMI_SyncVar.abErrorsTable[ERR_LoaderZSensorOutOfRange],
    bHead1VacuumError => sMMI_SyncVar.abErrorsTable[ERR_LoaderHead1Vacuum],
    bHead2VacuumError => sMMI_SyncVar.abErrorsTable[ERR_LoaderHead2Vacuum],
    bJackError => sMMI_SyncVar.abErrorsTable[ERR_LoaderJack],
    bXAxisError => sMMI_SyncVar.abErrorsTable[ERR_LoaderAxisX],
    bYAxisError => sMMI_SyncVar.abErrorsTable[ERR_LoaderAxisY],
    bZ1AxisError => sMMI_SyncVar.abErrorsTable[ERR_LoaderAxisZ1],
    bZ2AxisError => sMMI_SyncVar.abErrorsTable[ERR_LoaderAxisZ2],
    bTAxisError => sMMI_SyncVar.abErrorsTable[ERR_LoaderAxisTheta],
    bPlateVacuumError => sMMI_SyncVar.abErrorsTable[ERR_LoaderPlateVacuum],
    bActivateHead1Vacuum => QbLoaderActivateHead1Vacuum,
    bActivateHead1Blowing => QbLoaderActivateHead1Blowing,
    bActivateHead2Vacuum => QbLoaderActivateHead2Vacuum,
    bActivateHead2Blowing => QbLoaderActivateHead2Blowing,
    bActivatePlateVacuum => QbLoaderActivatePlateVacuum,
    bActivatePlateBlowing => QbLoaderActivatePlateBlowing,
    bMovePlateTakerUp => QbLoaderPlateTakerUp,
    bMovePlateTakerDown => QbLoaderPlateTakerDown,
    bAspirationBrushOn => bLoaderBrushAspirationOn,
    sOutGiveToTable => sGiversTakers.sLoaderTableGiverOut,
    sOutTakeFromTable => sGiversTakers.sLoaderTableTakerOut,
    sOutGiveToTurnOver => sGiversTakers.sLoaderTurnOverGiverOut,
    sOutTakeFromTurnOver => sGiversTakers.sLoaderTurnOverTakerOut,
    eRunStatus => sRunData.sStatusLoader,
    eVisionRunCmd => sRunData.eCmdVision,
    eLift1RunCmd => sRunData.eCmdLift1,
    eLift2RunCmd => sRunData.eCmdLift2,
    eRejectRunCmd => sRunData.eCmdReject,
    bVacuumInUse => bLoaderVacuumInUse,
    bManInterlockOut => bManInterlockLoaderLift,
    bManInterlockLiftOut => bManInterlockLoaderLift); // LoaderHdl

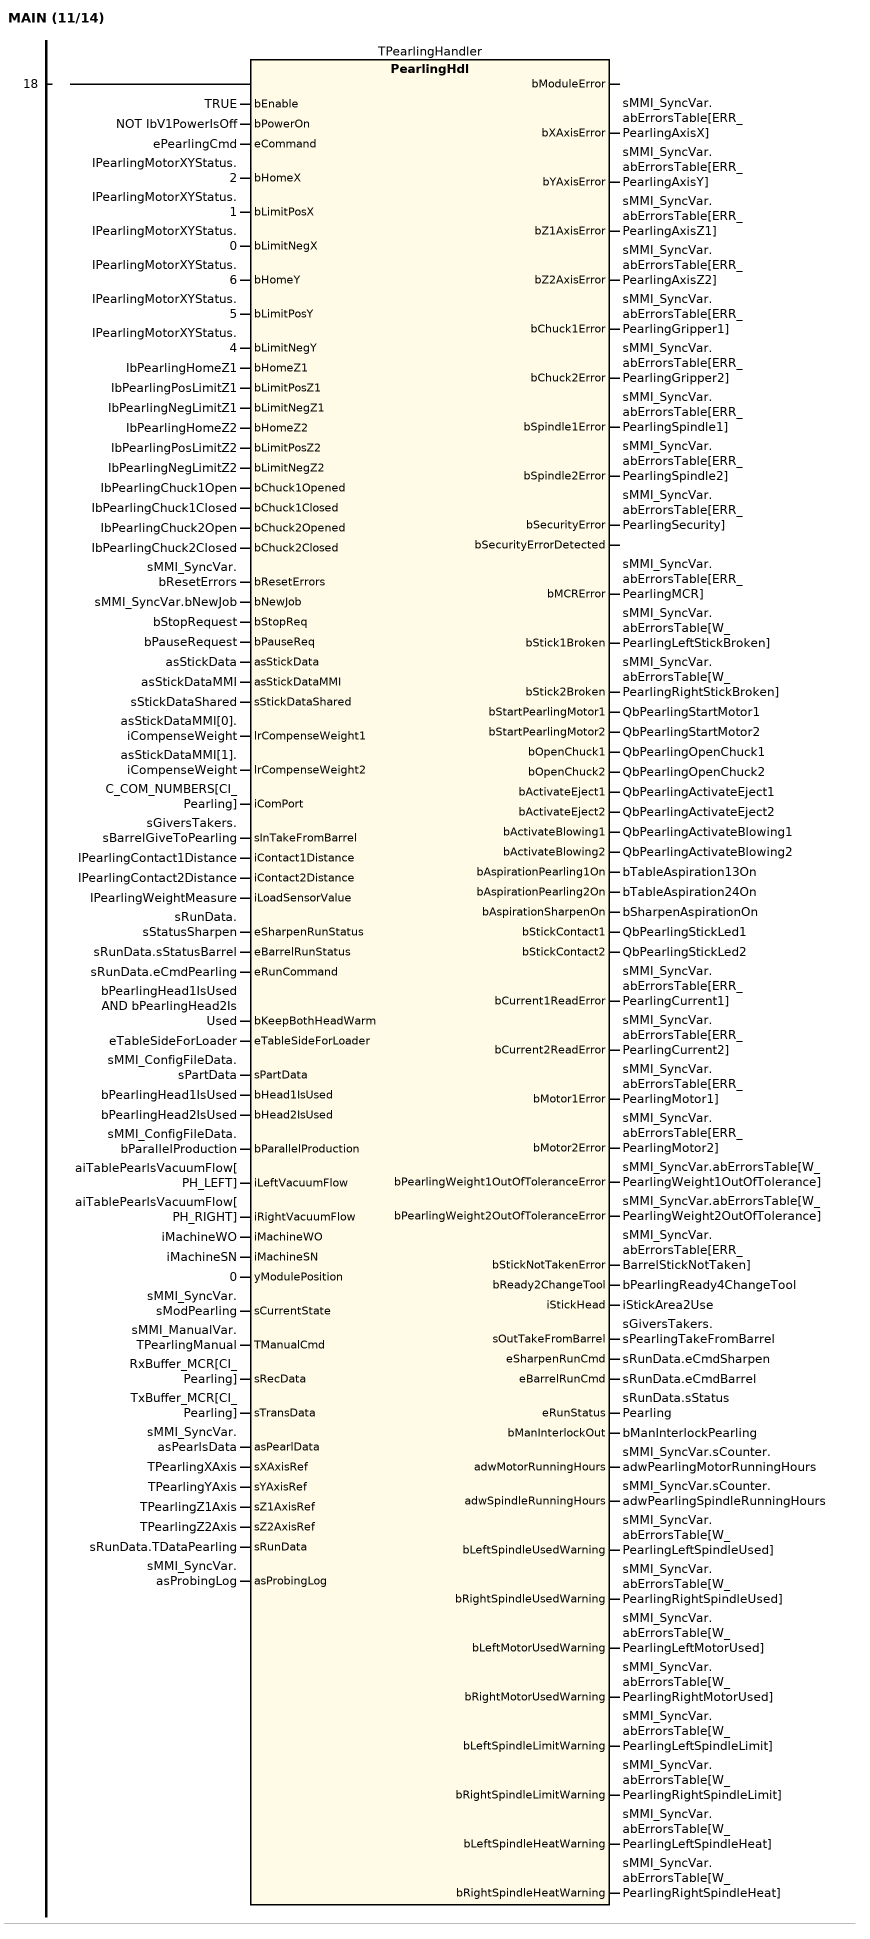
// NETWORK 18
TPearlingHandler(
    bEnable := TRUE,
    bPowerOn := NOT IbV1PowerIsOff,
    eCommand := ePearlingCmd,
    bHomeX := IPearlingMotorXYStatus.2,
    bLimitPosX := IPearlingMotorXYStatus.1,
    bLimitNegX := IPearlingMotorXYStatus.0,
    bHomeY := IPearlingMotorXYStatus.6,
    bLimitPosY := IPearlingMotorXYStatus.5,
    bLimitNegY := IPearlingMotorXYStatus.4,
    bHomeZ1 := IbPearlingHomeZ1,
    bLimitPosZ1 := IbPearlingPosLimitZ1,
    bLimitNegZ1 := IbPearlingNegLimitZ1,
    bHomeZ2 := IbPearlingHomeZ2,
    bLimitPosZ2 := IbPearlingPosLimitZ2,
    bLimitNegZ2 := IbPearlingNegLimitZ2,
    bChuck1Opened := IbPearlingChuck1Open,
    bChuck1Closed := IbPearlingChuck1Closed,
    bChuck2Opened := IbPearlingChuck2Open,
    bChuck2Closed := IbPearlingChuck2Closed,
    bResetErrors := sMMI_SyncVar.bResetErrors,
    bNewJob := sMMI_SyncVar.bNewJob,
    bStopReq := bStopRequest,
    bPauseReq := bPauseRequest,
    asStickData := asStickData,
    asStickDataMMI := asStickDataMMI,
    sStickDataShared := sStickDataShared,
    lrCompenseWeight1 := asStickDataMMI[0].iCompenseWeight,
    lrCompenseWeight2 := asStickDataMMI[1].iCompenseWeight,
    iComPort := C_COM_NUMBERS[CI_Pearling],
    sInTakeFromBarrel := sGiversTakers.sBarrelGiveToPearling,
    iContact1Distance := IPearlingContact1Distance,
    iContact2Distance := IPearlingContact2Distance,
    iLoadSensorValue := IPearlingWeightMeasure,
    eSharpenRunStatus := sRunData.sStatusSharpen,
    eBarrelRunStatus := sRunData.sStatusBarrel,
    eRunCommand := sRunData.eCmdPearling,
    bKeepBothHeadWarm := bPearlingHead1IsUsed AND bPearlingHead2IsUsed,
    eTableSideForLoader := eTableSideForLoader,
    sPartData := sMMI_ConfigFileData.sPartData,
    bHead1IsUsed := bPearlingHead1IsUsed,
    bHead2IsUsed := bPearlingHead2IsUsed,
    bParallelProduction := sMMI_ConfigFileData.bParallelProduction,
    iLeftVacuumFlow := aiTablePearlsVacuumFlow[PH_LEFT],
    iRightVacuumFlow := aiTablePearlsVacuumFlow[PH_RIGHT],
    iMachineWO := iMachineWO,
    iMachineSN := iMachineSN,
    yModulePosition := 0,
    sCurrentState := sMMI_SyncVar.sModPearling,
    TManualCmd := sMMI_ManualVar.TPearlingManual,
    sRecData := RxBuffer_MCR[CI_Pearling],
    sTransData := TxBuffer_MCR[CI_Pearling],
    asPearlData := sMMI_SyncVar.asPearlsData,
    sXAxisRef := TPearlingXAxis,
    sYAxisRef := TPearlingYAxis,
    sZ1AxisRef := TPearlingZ1Axis,
    sZ2AxisRef := TPearlingZ2Axis,
    sRunData := sRunData.TDataPearling,
    asProbingLog := sMMI_SyncVar.asProbingLog,
    bXAxisError => sMMI_SyncVar.abErrorsTable[ERR_PearlingAxisX],
    bYAxisError => sMMI_SyncVar.abErrorsTable[ERR_PearlingAxisY],
    bZ1AxisError => sMMI_SyncVar.abErrorsTable[ERR_PearlingAxisZ1],
    bZ2AxisError => sMMI_SyncVar.abErrorsTable[ERR_PearlingAxisZ2],
    bChuck1Error => sMMI_SyncVar.abErrorsTable[ERR_PearlingGripper1],
    bChuck2Error => sMMI_SyncVar.abErrorsTable[ERR_PearlingGripper2],
    bSpindle1Error => sMMI_SyncVar.abErrorsTable[ERR_PearlingSpindle1],
    bSpindle2Error => sMMI_SyncVar.abErrorsTable[ERR_PearlingSpindle2],
    bSecurityError => sMMI_SyncVar.abErrorsTable[ERR_PearlingSecurity],
    bMCRError => sMMI_SyncVar.abErrorsTable[ERR_PearlingMCR],
    bStick1Broken => sMMI_SyncVar.abErrorsTable[W_PearlingLeftStickBroken],
    bStick2Broken => sMMI_SyncVar.abErrorsTable[W_PearlingRightStickBroken],
    bStartPearlingMotor1 => QbPearlingStartMotor1,
    bStartPearlingMotor2 => QbPearlingStartMotor2,
    bOpenChuck1 => QbPearlingOpenChuck1,
    bOpenChuck2 => QbPearlingOpenChuck2,
    bActivateEject1 => QbPearlingActivateEject1,
    bActivateEject2 => QbPearlingActivateEject2,
    bActivateBlowing1 => QbPearlingActivateBlowing1,
    bActivateBlowing2 => QbPearlingActivateBlowing2,
    bAspirationPearling1On => bTableAspiration13On,
    bAspirationPearling2On => bTableAspiration24On,
    bAspirationSharpenOn => bSharpenAspirationOn,
    bStickContact1 => QbPearlingStickLed1,
    bStickContact2 => QbPearlingStickLed2,
    bCurrent1ReadError => sMMI_SyncVar.abErrorsTable[ERR_PearlingCurrent1],
    bCurrent2ReadError => sMMI_SyncVar.abErrorsTable[ERR_PearlingCurrent2],
    bMotor1Error => sMMI_SyncVar.abErrorsTable[ERR_PearlingMotor1],
    bMotor2Error => sMMI_SyncVar.abErrorsTable[ERR_PearlingMotor2],
    bPearlingWeight1OutOfToleranceError => sMMI_SyncVar.abErrorsTable[W_PearlingWeight1OutOfTolerance],
    bPearlingWeight2OutOfToleranceError => sMMI_SyncVar.abErrorsTable[W_PearlingWeight2OutOfTolerance],
    bStickNotTakenError => sMMI_SyncVar.abErrorsTable[ERR_BarrelStickNotTaken],
    bReady2ChangeTool => bPearlingReady4ChangeTool,
    iStickHead => iStickArea2Use,
    sOutTakeFromBarrel => sGiversTakers.sPearlingTakeFromBarrel,
    eSharpenRunCmd => sRunData.eCmdSharpen,
    eBarrelRunCmd => sRunData.eCmdBarrel,
    eRunStatus => sRunData.sStatusPearling,
    bManInterlockOut => bManInterlockPearling,
    adwMotorRunningHours => sMMI_SyncVar.sCounter.adwPearlingMotorRunningHours,
    adwSpindleRunningHours => sMMI_SyncVar.sCounter.adwPearlingSpindleRunningHours,
    bLeftSpindleUsedWarning => sMMI_SyncVar.abErrorsTable[W_PearlingLeftSpindleUsed],
    bRightSpindleUsedWarning => sMMI_SyncVar.abErrorsTable[W_PearlingRightSpindleUsed],
    bLeftMotorUsedWarning => sMMI_SyncVar.abErrorsTable[W_PearlingLeftMotorUsed],
    bRightMotorUsedWarning => sMMI_SyncVar.abErrorsTable[W_PearlingRightMotorUsed],
    bLeftSpindleLimitWarning => sMMI_SyncVar.abErrorsTable[W_PearlingLeftSpindleLimit],
    bRightSpindleLimitWarning => sMMI_SyncVar.abErrorsTable[W_PearlingRightSpindleLimit],
    bLeftSpindleHeatWarning => sMMI_SyncVar.abErrorsTable[W_PearlingLeftSpindleHeat],
    bRightSpindleHeatWarning => sMMI_SyncVar.abErrorsTable[W_PearlingRightSpindleHeat]); // PearlingHdl

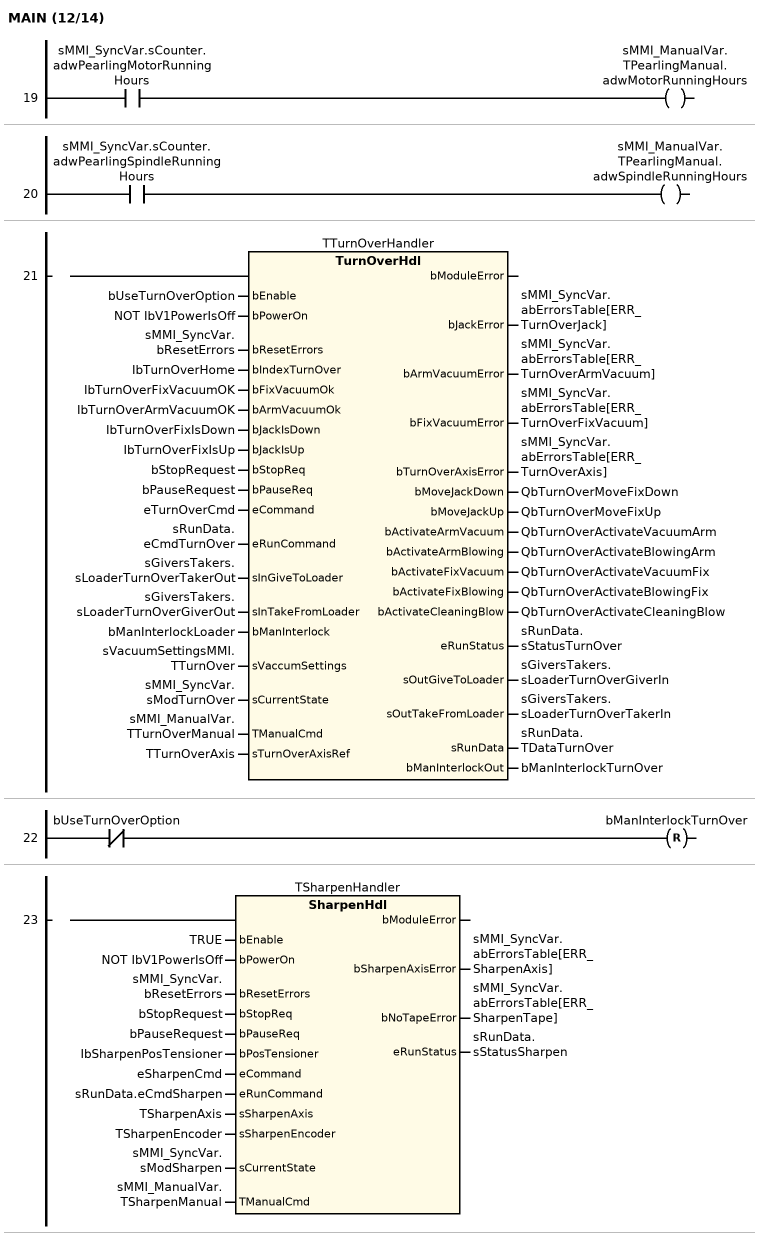
// NETWORK 19
sMMI_ManualVar.TPearlingManual.adwMotorRunningHours := sMMI_SyncVar.sCounter.adwPearlingMotorRunningHours;

// NETWORK 20
sMMI_ManualVar.TPearlingManual.adwSpindleRunningHours := sMMI_SyncVar.sCounter.adwPearlingSpindleRunningHours;

// NETWORK 21
TTurnOverHandler(
    bEnable := bUseTurnOverOption,
    bPowerOn := NOT IbV1PowerIsOff,
    bResetErrors := sMMI_SyncVar.bResetErrors,
    bIndexTurnOver := IbTurnOverHome,
    bFixVacuumOk := IbTurnOverFixVacuumOK,
    bArmVacuumOk := IbTurnOverArmVacuumOK,
    bJackIsDown := IbTurnOverFixIsDown,
    bJackIsUp := IbTurnOverFixIsUp,
    bStopReq := bStopRequest,
    bPauseReq := bPauseRequest,
    eCommand := eTurnOverCmd,
    eRunCommand := sRunData.eCmdTurnOver,
    sInGiveToLoader := sGiversTakers.sLoaderTurnOverTakerOut,
    sInTakeFromLoader := sGiversTakers.sLoaderTurnOverGiverOut,
    bManInterlock := bManInterlockLoader,
    sVaccumSettings := sVacuumSettingsMMI.TTurnOver,
    sCurrentState := sMMI_SyncVar.sModTurnOver,
    TManualCmd := sMMI_ManualVar.TTurnOverManual,
    sTurnOverAxisRef := TTurnOverAxis,
    bJackError => sMMI_SyncVar.abErrorsTable[ERR_TurnOverJack],
    bArmVacuumError => sMMI_SyncVar.abErrorsTable[ERR_TurnOverArmVacuum],
    bFixVacuumError => sMMI_SyncVar.abErrorsTable[ERR_TurnOverFixVacuum],
    bTurnOverAxisError => sMMI_SyncVar.abErrorsTable[ERR_TurnOverAxis],
    bMoveJackDown => QbTurnOverMoveFixDown,
    bMoveJackUp => QbTurnOverMoveFixUp,
    bActivateArmVacuum => QbTurnOverActivateVacuumArm,
    bActivateArmBlowing => QbTurnOverActivateBlowingArm,
    bActivateFixVacuum => QbTurnOverActivateVacuumFix,
    bActivateFixBlowing => QbTurnOverActivateBlowingFix,
    bActivateCleaningBlow => QbTurnOverActivateCleaningBlow,
    eRunStatus => sRunData.sStatusTurnOver,
    sOutGiveToLoader => sGiversTakers.sLoaderTurnOverGiverIn,
    sOutTakeFromLoader => sGiversTakers.sLoaderTurnOverTakerIn,
    sRunData => sRunData.TDataTurnOver,
    bManInterlockOut => bManInterlockTurnOver); // TurnOverHdl

// NETWORK 22
bManInterlockTurnOver R= NOT bUseTurnOverOption;

// NETWORK 23
TSharpenHandler(
    bEnable := TRUE,
    bPowerOn := NOT IbV1PowerIsOff,
    bResetErrors := sMMI_SyncVar.bResetErrors,
    bStopReq := bStopRequest,
    bPauseReq := bPauseRequest,
    bPosTensioner := IbSharpenPosTensioner,
    eCommand := eSharpenCmd,
    eRunCommand := sRunData.eCmdSharpen,
    sSharpenAxis := TSharpenAxis,
    sSharpenEncoder := TSharpenEncoder,
    sCurrentState := sMMI_SyncVar.sModSharpen,
    TManualCmd := sMMI_ManualVar.TSharpenManual,
    bSharpenAxisError => sMMI_SyncVar.abErrorsTable[ERR_SharpenAxis],
    bNoTapeError => sMMI_SyncVar.abErrorsTable[ERR_SharpenTape],
    eRunStatus => sRunData.sStatusSharpen); // SharpenHdl

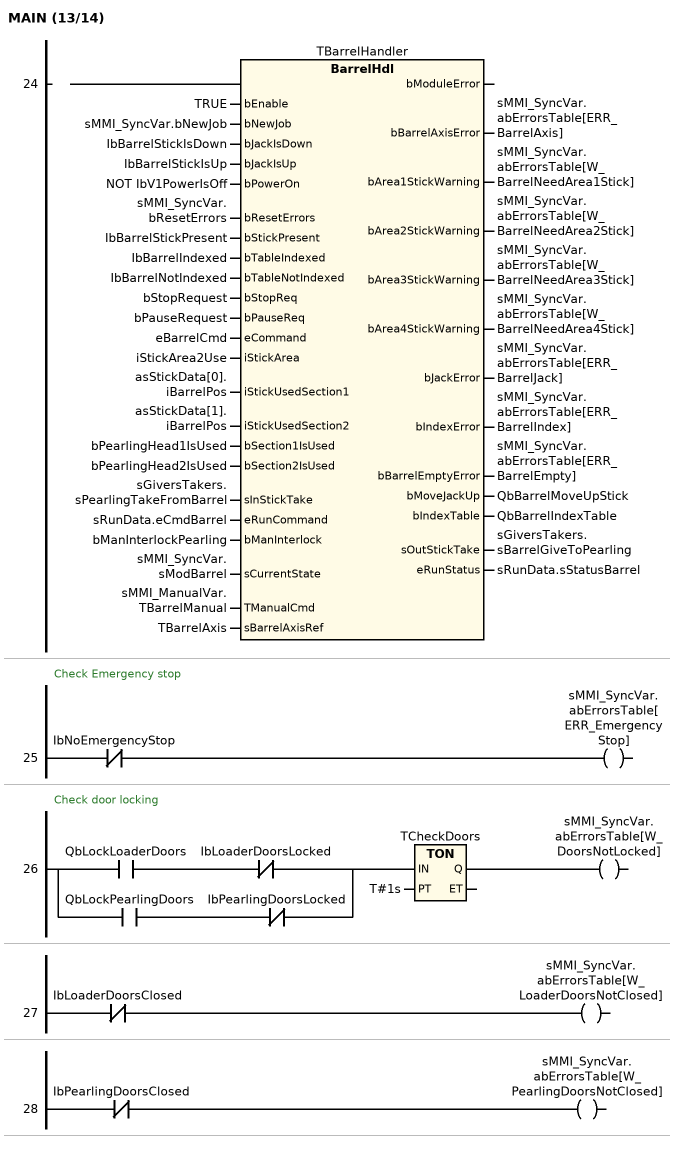
// NETWORK 24
TBarrelHandler(
    bEnable := TRUE,
    bNewJob := sMMI_SyncVar.bNewJob,
    bJackIsDown := IbBarrelStickIsDown,
    bJackIsUp := IbBarrelStickIsUp,
    bPowerOn := NOT IbV1PowerIsOff,
    bResetErrors := sMMI_SyncVar.bResetErrors,
    bStickPresent := IbBarrelStickPresent,
    bTableIndexed := IbBarrelIndexed,
    bTableNotIndexed := IbBarrelNotIndexed,
    bStopReq := bStopRequest,
    bPauseReq := bPauseRequest,
    eCommand := eBarrelCmd,
    iStickArea := iStickArea2Use,
    iStickUsedSection1 := asStickData[0].iBarrelPos,
    iStickUsedSection2 := asStickData[1].iBarrelPos,
    bSection1IsUsed := bPearlingHead1IsUsed,
    bSection2IsUsed := bPearlingHead2IsUsed,
    sInStickTake := sGiversTakers.sPearlingTakeFromBarrel,
    eRunCommand := sRunData.eCmdBarrel,
    bManInterlock := bManInterlockPearling,
    sCurrentState := sMMI_SyncVar.sModBarrel,
    TManualCmd := sMMI_ManualVar.TBarrelManual,
    sBarrelAxisRef := TBarrelAxis,
    bBarrelAxisError => sMMI_SyncVar.abErrorsTable[ERR_BarrelAxis],
    bArea1StickWarning => sMMI_SyncVar.abErrorsTable[W_BarrelNeedArea1Stick],
    bArea2StickWarning => sMMI_SyncVar.abErrorsTable[W_BarrelNeedArea2Stick],
    bArea3StickWarning => sMMI_SyncVar.abErrorsTable[W_BarrelNeedArea3Stick],
    bArea4StickWarning => sMMI_SyncVar.abErrorsTable[W_BarrelNeedArea4Stick],
    bJackError => sMMI_SyncVar.abErrorsTable[ERR_BarrelJack],
    bIndexError => sMMI_SyncVar.abErrorsTable[ERR_BarrelIndex],
    bBarrelEmptyError => sMMI_SyncVar.abErrorsTable[ERR_BarrelEmpty],
    bMoveJackUp => QbBarrelMoveUpStick,
    bIndexTable => QbBarrelIndexTable,
    sOutStickTake => sGiversTakers.sBarrelGiveToPearling,
    eRunStatus => sRunData.sStatusBarrel); // BarrelHdl

// NETWORK 25
// Check Emergency stop
sMMI_SyncVar.abErrorsTable[ERR_EmergencyStop] := NOT IbNoEmergencyStop;

// NETWORK 26
// Check door locking
TCheckDoors(IN := QbLockLoaderDoors AND NOT IbLoaderDoorsLocked OR QbLockPearlingDoors AND NOT IbPearlingDoorsLocked, PT := T#1s); // TON
sMMI_SyncVar.abErrorsTable[W_DoorsNotLocked] := TCheckDoors.Q;

// NETWORK 27
sMMI_SyncVar.abErrorsTable[W_LoaderDoorsNotClosed] := NOT IbLoaderDoorsClosed;

// NETWORK 28
sMMI_SyncVar.abErrorsTable[W_PearlingDoorsNotClosed] := NOT IbPearlingDoorsClosed;

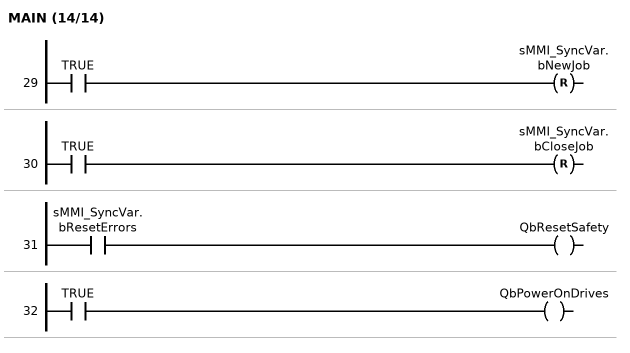
// NETWORK 29
sMMI_SyncVar.bNewJob R= TRUE;

// NETWORK 30
sMMI_SyncVar.bCloseJob R= TRUE;

// NETWORK 31
QbResetSafety := sMMI_SyncVar.bResetErrors;

// NETWORK 32
QbPowerOnDrives := TRUE;

END_PROGRAM

(* stored: Version 1.1.0.1, ProductVersion 3.1.4022.18
   POU MAIN: Id {ba02f46c-bfeb-417b-ac69-8e7d94efd5af}, SpecialFunc None *)
